PROGRAM MAIN
VAR_OUTPUT
    timerValue0: TIME;
    timerValue1: TIME;
END_VAR
VAR
    cnt: LINT;
    first: BOOL := TRUE;
    curTimerValue: TIME;
    state0: STATE;
    curTime: LREAL;
    loopsKilled: LINT;
END_VAR
VAR_TEMP
    lastTimerValue: TIME;
    curDeltaTime: TIME;
    curDeltaSecs: LREAL;
    state1: STATE;
    progress: BOOL;
    loopCount: INT;
END_VAR


// Handle 'time' and cycle time.
cnt := cnt + 1;

timer0(IN := curTimer = 0, PT := T#1D);
timer1(IN := curTimer = 1, PT := T#1D);
timerValue0 := timer0.ET;
timerValue1 := timer1.ET;

lastTimerValue := curTimerValue;
IF curTimer = 0 THEN
    curTimerValue := timerValue0;
ELSE
    curTimerValue := timerValue1;
END_IF;
curDeltaTime := curTimerValue - lastTimerValue;
curDeltaSecs := TIME_TO_LREAL(curDeltaTime) / 1000;
curTime := curTime + curDeltaSecs;

IF cnt MOD 10 = 0 THEN
    curTimer := 1 - curTimer;
    curTimerValue := T#0S;
    timer0(IN := curTimer = 0, PT := T#1D);
    timer1(IN := curTimer = 1, PT := T#1D);
    timerValue0 := timer0.ET;
    timerValue1 := timer1.ET;
END_IF;

IF first THEN
    first := FALSE;

    // Initialize state variables for initial state.
    state0.dvar_M_p_x := 1;
    state0.dvar_M_p := elit_l1;
    state0.dvar_M_q_y := 2;
    state0.dvar_M_q_b := FALSE;
ELSE
    // Update continuous variables for time delay.

    state0.curTime := curTime;
END_IF;

// Event loop.
WHILE TRUE DO
    progress := FALSE;

    // Event "e".
    IF NOT progress THEN
        IF (state0.dvar_M_p) = (elit_l1) THEN
            progress := TRUE;
            state1 := state0;

            state1.dvar_M_p_x := (state0.dvar_M_q_y) + (1);
            state1.dvar_M_p := elit_l2;
            state1.dvar_M_q_y := (state0.dvar_M_p_x) + (1);

            state0 := state1;
        END_IF;
    END_IF;

    // Event "f".
    IF NOT progress THEN
        IF state0.dvar_M_q_b THEN
            progress := TRUE;
            state1 := state0;

            IF ((state0.dvar_M_q_y) < (6)) THEN
                state1.dvar_M_q_y := (state0.dvar_M_q_y) + (1);
            ELSE
                state1.dvar_M_q_b := NOT(state0.dvar_M_q_b);
            END_IF;

            state0 := state1;
        END_IF;
    END_IF;

    // Event "tau".
    IF NOT progress THEN
        IF (state0.dvar_M_q_y) < (6) THEN
            progress := TRUE;
            state1 := state0;

            state1.dvar_M_q_y := (state0.dvar_M_q_y) + (1);

            state0 := state1;
        END_IF;
    END_IF;

    // Done with events?
    IF NOT progress THEN
        EXIT;
    END_IF;

    // Protect against events that are always enabled.
    loopCount := loopCount + 1;
    IF loopCount >= 100 THEN
        loopsKilled := loopsKilled + 1;
        EXIT;
    END_IF;
END_WHILE;

END_PROGRAM

(* stored: ProductVersion 3.1.0.18, Version 1.1.0.1 *)
